// TwinCAT 3 PLC project PLC
// ProgramVersion: 3.1.4024.0
// libraries:
//   Tc2_EtherCAT, * (Beckhoff Automation GmbH)
//   Tc2_Standard, * (Beckhoff Automation GmbH)
//   Tc2_System, * (Beckhoff Automation GmbH)
//   Tc3_Module, * (Beckhoff Automation GmbH)
//   VisuDialogs, * (System)
// project tree:
//   DUTs/ ST_3D_Values.TcDUT
//   / GlobalTextList.TcGTLO, PlcTask.TcTTO, Visualisierungsmanager.TcVMO (not stored)
//   GVLs/ GVL_SensorFusion.TcGVL
//   POUs/Filter/ FB_ComplementaryFilter.TcPOU, FB_KalmanFilter.TcPOU, FB_MadgwickFilter.TcPOU, FB_MahonyFilter.TcPOU, FB_MovingAverageFilter.TcPOU (not stored), FB_MovingAverageFilter_3D.TcPOU
//   POUs/Filter/obsolete/ FBiFilter.TcPOU (not stored), FB_Complementary_Ex.TcPOU
//   POUs/Helping Functions/ ATAN2.TcPOU, ATAN2_deg.TcPOU
//   POUs/Helping Functions/obsolete/ iGetNextBufferPointer.TcPOU, iGetPriorBufferPointer.TcPOU
//   POUs/ MAIN.TcPOU
//   VISUs/ Visualization.TcVIS
// real-time tasks:
//   TASK PlcTask: cycle T#250us, priority 20, ADS port 350
// I/O:
//   DEVICE Device 3 (EtherCAT) (disabled), AmsNetId 172.17.129.121.4.1
//     Box 1 (EP3751-0260) [EP3751-0260 Acceleration Sensor and Gyroscope]
// variable links:
//   PLC/PLC Instance <-> Device 3 (EtherCAT)/Box 1 (EP3751-0260)
//     PlcTask Inputs/MAIN.stAccAxis/X <-> AI Acc X Samples 1 (Real32)/Samples[0]
//     PlcTask Inputs/MAIN.stAccAxis/Y <-> AI Acc Y Samples 1 (Real32)/Samples[0]
//     PlcTask Inputs/MAIN.stAccAxis/Z <-> AI Acc Z Samples 1 (Real32)/Samples[0]
//     PlcTask Inputs/MAIN.stGyroAxis/X <-> AI Gyro X Samples 1 (Real32)/Samples[0]
//     PlcTask Inputs/MAIN.stGyroAxis/Y <-> AI Gyro Y Samples 1 (Real32)/Samples[0]
//     PlcTask Inputs/MAIN.stGyroAxis/Z <-> AI Gyro Z Samples 1 (Real32)/Samples[0]

CONFIGURATION PLC
    RESOURCE PLC ON TwinCAT3
        TASK PlcTask(INTERVAL := T#250us, PRIORITY := 20);
        PROGRAM MAIN WITH PlcTask : MAIN;
    END_RESOURCE
END_CONFIGURATION

// ---- DUTs/ST_3D_Values.TcDUT
TYPE ST_3D_Values :
STRUCT
	X :REAL;
	Y :REAL;
	Z :REAL;
END_STRUCT
END_TYPE

// ---- GVLs/GVL_SensorFusion.TcGVL
{attribute 'qualified_only'}
VAR_GLOBAL CONSTANT
	buffersize_filter :UINT :=2000;
END_VAR

// ---- POUs/MAIN.TcPOU
PROGRAM MAIN
VAR
	stGyroAxis AT %I* : ST_3d_values;
	stcorrAxis : ST_3d_values;
	stOffset	:ST_3d_values;

	fbMovingAverage_3D: FB_MovingAverageFilter_3D;
	a_fBuffer : ARRAY[0..2] OF ARRAY[ 0..GVL_SensorFusion.buffersize_filter-1] OF REAL;
	
(* Accelerometer values *)
	stAccAxis AT %I* : ST_3d_values;
	normalizedAcceleration : ARRAY [0..2] OF LREAL;

(* Working variables *)
	fbStartOffsetCalibration : R_TRIG;
	bReset: BOOL;
	fbOffsetSet : R_TRIG;
	bResetAngles: BOOL;

	fCycleTime 				: LREAL; // PLC cycle time in s (has to match with ODR of sensor => for prototype this is static 4000Hz)
	nTaskIndex				: DINT;
	bReady					: BOOL;
	
(*Disclaimer: This is a sample still in prototype phase.
Please be aware that functionalities/ PDOs / CoEs can differ in series variant.
*)
	fbKalmanFilter:FB_KalmanFilter;
	fbMadgwickFilter:FB_MadgwickFilter;
	fbComplementaryFilter:FB_ComplementaryFilter;
	fbMahonyFilter:FB_MahonyFilter;
	stEulerAngle_Gyro:ST_3D_Values;
END_VAR

nTaskIndex:=GETCURTASKINDEXEX();
IF nTaskIndex>0 THEN
	fCycletime:=UDINT_TO_LREAL(_TaskInfo[GETCURTASKINDEXEX()].CycleTime) / 10_000_000;
END_IF

// get Sensoroffset
fbStartOffsetCalibration(clk:=bReset);

fbMovingAverage_3D( stSampleData:=stGyroAxis, bEnable:=NOT fbStartOffsetCalibration.Q, a_fSamples:=a_fBuffer);
fbOffsetSet(clk:=fbMovingAverage_3D.bBufferFilledX);
IF fbOffsetSet.Q THEN
	stOffset.x:=fbMovingAverage_3D.stAvgData.X;
	stOffset.y:=fbMovingAverage_3D.stAvgData.y;
	stOffset.z:=fbMovingAverage_3D.stAvgData.z;
	stEulerAngle_Gyro.x:=0;
	stEulerAngle_Gyro.y:=0;
	stEulerAngle_Gyro.z:=0;
ELSIF bResetAngles THEN
	stEulerAngle_Gyro.x:=0;
	stEulerAngle_Gyro.y:=0;
	stEulerAngle_Gyro.z:=0;
	bResetAngles:=FALSE;
END_IF

bReady:=fbMovingAverage_3D.bBufferFilledX;

//correct Gyro-Values with Offset
stcorrAxis.X:= stGyroAxis.X - stOffset.x;
stcorrAxis.Y:= stGyroAxis.Y - stOffset.y;
stcorrAxis.Z:= stGyroAxis.Z - stOffset.z;


	//Calculate Euler Angles by Sensorfusion
	fbKalmanFilter(
		stAccelData:= stAccAxis, 
		stGyroData:= stcorrAxis,  
		fCycleTime:= fCycletime,
		bSetReference:=fbMovingAverage_3D.bBufferFilledX );
		
	fbMadgwickFilter(
		stAccelData:= stAccAxis, 
		stGyroData:= stcorrAxis,  
		fcycletime:=fCycletime , 
		bSetReference:= fbMovingAverage_3D.bBufferFilledX );
		
	fbComplementaryFilter(
		stAccelData:= stAccAxis, 
		stGyroData:= stcorrAxis,  
		fcycletime:=fCycletime , 
		bSetReference:= fbMovingAverage_3D.bBufferFilledX );
		
	fbMahonyFilter(
		stAccelData:= stAccAxis, 
		stGyroData:= stcorrAxis,  
		fcycletime:=fCycletime , 
		bSetReference:= fbMovingAverage_3D.bBufferFilledX );
		
stEulerAngle_Gyro.x := stEulerAngle_Gyro.x + stcorrAxis.x * fCycleTime;
stEulerAngle_Gyro.y := stEulerAngle_Gyro.y + stcorrAxis.y * fCycleTime;
stEulerAngle_Gyro.z := stEulerAngle_Gyro.z + stcorrAxis.Z * fCycleTime;

END_PROGRAM

// ---- POUs/Filter/FB_MovingAverageFilter_3D.TcPOU
FUNCTION_BLOCK FB_MovingAverageFilter_3D
VAR_INPUT
    stSampleData : ST_3D_values; // New Data in 3 axes
    nNumSamples : UINT:= gvl_sensorFusion.buffersize_filter;              // Number of samples for the moving average
    bEnable 	: BOOL;                   // Execute flag
END_VAR

VAR_OUTPUT
    stAvgData : ST_3D_values; // New Data in 3 axes
    bBufferFilledX : BOOL;            // Flag indicating if the buffer for X axis is filled
    bBufferFilledY : BOOL;            // Flag indicating if the buffer for Y axis is filled
    bBufferFilledZ : BOOL;            // Flag indicating if the buffer for Z axis is filled
END_VAR

VAR_IN_OUT
    a_fSamples : ARRAY[0..2] OF ARRAY[ 0..GVL_SensorFusion.buffersize_filter-1] OF REAL; // Array of arrays to store samples for three axes
END_VAR

VAR
	fbExecuteTrigger:r_trig;
	bInit:BOOL;
    fbMovingAverageX : FB_MovingAverageFilter; // Instance for X axis
    fbMovingAverageY : FB_MovingAverageFilter; // Instance for Y axis
    fbMovingAverageZ : FB_MovingAverageFilter; // Instance for Z axis
END_VAR

IF NOT bEnable THEN
	bInit:=bInit;
END_IF

fbMovingAverageX(
    fInputValue := stSampleData.X,
    nNumSamples := nNumSamples,
    bEnable := bEnable,
    fAvgValue => stAvgData.x,
    bBufferFilled => bBufferFilledX,
    a_fSamples := a_fSamples[0]
);

fbMovingAverageY(
    fInputValue := stSampleData.y,
    nNumSamples := nNumSamples,
    bEnable := bEnable,
    fAvgValue => stAvgData.y,
    bBufferFilled => bBufferFilledY,
    a_fSamples := a_fSamples[1]
);

fbMovingAverageZ(
    fInputValue := stSampleData.z,
    nNumSamples := nNumSamples,
    bEnable := bEnable,
    fAvgValue => stAvgData.z,
    bBufferFilled => bBufferFilledZ,
    a_fSamples := a_fSamples[2]
);

END_FUNCTION_BLOCK

// ---- POUs/Filter/FB_KalmanFilter.TcPOU
FUNCTION_BLOCK FB_KalmanFilter
VAR_INPUT
    stAccelData : ST_3D_values; // Acceleration Data in (g)
    stGyroData : ST_3D_values; // Gyroscope Data in (°/s)
	fCycleTime: REAL; 			// CycleTime of sensor data in s
	fQ_angle : REAL := 0.001;     // Process noise variance for the angle
    fQ_bias : REAL := 0.003;      // Process noise variance for the bias
    fR_measure : REAL := 0.03;    // Measurement noise variance
    bSetReference : BOOL := FALSE; // Flag to set the current position as the reference position
END_VAR
VAR_OUTPUT
    stEulerAngle_deg : ST_3D_values; // Estimated Euler angle in degrees X= Pitch, Y=Roll, Z=Yaw
    stEulerAngle_rad : ST_3D_values; // Estimated Euler angle in rad X= Pitch, Y=Roll, Z=Yaw
END_VAR
VAR
	// Reference angles
	stRef_Angles_deg :ST_3d_values; // Reference orientation (bSetReference; angles in degrees)
	
    // Variables for X-axis
    fAngle_prevX_rad : LREAL := 0.0;   // Previous angle for X-axis in radians
    fBiasX : LREAL := 0.0;             // Gyroscope bias for X-axis
    fRateX : LREAL := 0.0;             // Rate of change of the angle for X-axis

    fP_00X : LREAL := 1.0;             // Covariance matrix for X-axis
    fP_01X : LREAL := 0.0;
    fP_10X : LREAL := 0.0;
    fP_11X : LREAL := 1.0;

    fY_X : LREAL;                      // Angle difference for X-axis
    fS_X : LREAL;                      // Estimate error for X-axis
    fK_0X : LREAL;                     // Kalman gain for X-axis
    fK_1X : LREAL;                     // Kalman gain for X-axis

    // Variables for Y-axis
    fAngle_prevY_rad : LREAL := 0.0;   // Previous angle for Y-axis in radians
    fBiasY : LREAL := 0.0;             // Gyroscope bias for Y-axis
    fRateY : LREAL := 0.0;             // Rate of change of the angle for Y-axis

    fP_00Y : LREAL := 1.0;             // Covariance matrix for Y-axis
    fP_01Y : LREAL := 0.0;
    fP_10Y : LREAL := 0.0;
    fP_11Y : LREAL := 1.0;

    fY_Y : LREAL;                      // Angle difference for Y-axis
    fS_Y : LREAL;                      // Estimate error for Y-axis
    fK_0Y : LREAL;                     // Kalman gain for Y-axis
    fK_1Y : LREAL;                     // Kalman gain for Y-axis

    // Variables for Z-axis
    fAngle_prevZ_rad : LREAL := 0.0;   // Previous angle for Z-axis in radians
    fBiasZ : LREAL := 0.0;             // Gyroscope bias for Z-axis
    fRateZ : LREAL := 0.0;             // Rate of change of the angle for Z-axis

    fP_00Z : LREAL := 1.0;             // Covariance matrix for Z-axis
    fP_01Z : LREAL := 0.0;
    fP_10Z : LREAL := 0.0;
    fP_11Z : LREAL := 1.0;

    fY_Z : LREAL;                      // Angle difference for Z-axis
    fS_Z : LREAL;                      // Estimate error for Z-axis
    fK_0Z : LREAL;                     // Kalman gain for Z-axis
    fK_1Z : LREAL;                     // Kalman gain for Z-axis
	
	// Convert accelerometer data to angles (pitch, roll) in radians
    fPitchAccel_rad : LREAL;
    fRollAccel_rad : LREAL;
	
	fbSetReference: r_trig;
END_VAR

// Calculate accelerometer angles using ATAN2, which returns radians
IF (stAccelData.X * stAccelData.X + stAccelData.Z * stAccelData.Z > 0.0) THEN 
    fPitchAccel_rad := ATAN(stAccelData.Y / SQRT(stAccelData.X * stAccelData.X + stAccelData.Z * stAccelData.Z));
END_IF
IF (stAccelData.Y * stAccelData.Y + stAccelData.Z * stAccelData.Z > 0.0) THEN 
    fRollAccel_rad := ATAN(stAccelData.X / SQRT(stAccelData.Y * stAccelData.Y + stAccelData.Z * stAccelData.Z));
END_IF

// Prediction step for X-axis (Pitch)
fRateX := stGyroData.X - fBiasX;
fAngle_prevX_rad := fAngle_prevX_rad + fCycleTime * fRateX * PI / 180.0; // Conversion of rate from degrees/second to radians/second

fP_00X := fP_00X + fCycleTime * (fCycleTime * fP_11X - fP_01X - fP_10X + fQ_angle);
fP_01X := fP_01X - fCycleTime * fP_11X;
fP_10X := fP_10X - fCycleTime * fP_11X;
fP_11X := fP_11X + fQ_bias * fCycleTime;

// Measurement update for X-axis (Pitch)
fY_X := fPitchAccel_rad - fAngle_prevX_rad; // Using the pitch angle in radians
fS_X := fP_00X + fR_measure;
fK_0X := fP_00X / fS_X;
fK_1X := fP_10X / fS_X;

fAngle_prevX_rad := fAngle_prevX_rad + fK_0X * fY_X;
fBiasX := fBiasX + fK_1X * fY_X;

fP_00X := fP_00X - fK_0X * fP_00X;
fP_01X := fP_01X - fK_0X * fP_01X;
fP_10X := fP_10X - fK_1X * fP_00X;
fP_11X := fP_11X - fK_1X * fP_01X;

// Prediction step for Y-axis (Roll)
fRateY := stGyroData.Y - fBiasY;
fAngle_prevY_rad := fAngle_prevY_rad + fCycleTime * fRateY * PI / 180.0; // Conversion of rate from degrees/second to radians/second

fP_00Y := fP_00Y + fCycleTime * (fCycleTime * fP_11Y - fP_01Y - fP_10Y + fQ_angle);
fP_01Y := fP_01Y - fCycleTime * fP_11Y;
fP_10Y := fP_10Y - fCycleTime * fP_11Y;
fP_11Y := fP_11Y + fQ_bias * fCycleTime;

// Measurement update for Y-axis (Roll)
fY_Y := fRollAccel_rad - fAngle_prevY_rad; // Using the roll angle in radians
fS_Y := fP_00Y + fR_measure;
fK_0Y := fP_00Y / fS_Y;
fK_1Y := fP_10Y / fS_Y;

fAngle_prevY_rad := fAngle_prevY_rad + fK_0Y * fY_Y;
fBiasY := fBiasY + fK_1Y * fY_Y;

fP_00Y := fP_00Y - fK_0Y * fP_00Y;
fP_01Y := fP_01Y - fK_0Y * fP_01Y;
fP_10Y := fP_10Y - fK_1Y * fP_00Y;
fP_11Y := fP_11Y - fK_1Y * fP_01Y;

// Prediction step for Z-axis (Yaw)
fRateZ := stGyroData.Z - fBiasZ;
fAngle_prevZ_rad := fAngle_prevZ_rad + fCycleTime * fRateZ * PI / 180.0; // Conversion of rate from degrees/second to radians/second

fP_00Z := fP_00Z + fCycleTime * (fCycleTime * fP_11Z - fP_01Z - fP_10Z + fQ_angle);
fP_01Z := fP_01Z - fCycleTime * fP_11Z;
fP_10Z := fP_10Z - fCycleTime * fP_11Z;
fP_11Z := fP_11Z + fQ_bias * fCycleTime;

// Measurement update for Z-axis (Yaw)
// Since the accelerometer does not provide a direct yaw measurement, we use gyroscope data for the yaw update.
fY_Z := fRateZ; // Gyroscope rate in degrees/second
fS_Z := fP_00Z + fR_measure;
fK_0Z := fP_00Z / fS_Z;
fK_1Z := fP_10Z / fS_Z;

fAngle_prevZ_rad := fAngle_prevZ_rad + fK_0Z * fY_Z * fCycleTime * PI / 180.0; // Updating the yaw angle with gyroscope data and conversion to radians
fBiasZ := fBiasZ + fK_1Z * fY_Z * fCycleTime * PI / 180.0;

fP_00Z := fP_00Z - fK_0Z * fP_00Z;
fP_01Z := fP_01Z - fK_0Z * fP_01Z;
fP_10Z := fP_10Z - fK_1Z * fP_00Z;
fP_11Z := fP_11Z - fK_1Z * fP_01Z;

// Convert radians to degrees for output
stEulerAngle_deg.X := fAngle_prevX_rad * 180.0 / PI;
stEulerAngle_deg.Y := fAngle_prevY_rad * 180.0 / PI;
stEulerAngle_deg.Z := fAngle_prevZ_rad * 180.0 / PI;

fbSetReference(clk:=bSetReference);
// Set reference position if flag is active
IF fbSetReference.q THEN
    stRef_Angles_deg.X := stEulerAngle_deg.X;
    stRef_Angles_deg.Y := stEulerAngle_deg.Y;
    stRef_Angles_deg.Z := stEulerAngle_deg.Z;
END_IF

// Apply reference position
stEulerAngle_deg.X := stEulerAngle_deg.X - (stRef_Angles_deg.X);
stEulerAngle_deg.Y := stEulerAngle_deg.Y - (stRef_Angles_deg.Y);
stEulerAngle_deg.Z := stEulerAngle_deg.Z - (stRef_Angles_deg.Z);

stEulerAngle_rad.X := fAngle_prevX_rad - (stRef_Angles_deg.X) * PI / 180.0;
stEulerAngle_rad.Y := fAngle_prevY_rad - (stRef_Angles_deg.Y) * PI / 180.0;
stEulerAngle_rad.Z := fAngle_prevZ_rad - (stRef_Angles_deg.Z) * PI / 180.0;

END_FUNCTION_BLOCK

// ---- POUs/Filter/FB_MadgwickFilter.TcPOU
FUNCTION_BLOCK FB_MadgwickFilter
VAR_INPUT
    stAccelData : ST_3D_values; // Acceleration Data in (g)
    stGyroData : ST_3D_values; // Gyroscope Data in (°/s)
    fBeta: REAL := 0.05; // Algorithm gain
    fCycletime: REAL; // Time step (s)
    bSetReference: BOOL; // Flag to set reference position
END_VAR

VAR_OUTPUT
	fQ0 : LREAL := 1.0; // Quaternion component
    fQ1 : LREAL := 0.0; // Quaternion component
    fQ2 : LREAL := 0.0; // Quaternion component
    fQ3 : LREAL := 0.0; // Quaternion component
    stEulerAngle_deg : ST_3D_values; // Estimated Euler angle in degrees X= Pitch, Y=Roll, Z=Yaw
    stEulerAngle_rad : ST_3D_values; // Estimated Euler angle in rad X= Pitch, Y=Roll, Z=Yaw
END_VAR

VAR

	// Reference angles
	stRef_Angles_deg :ST_3d_values; // Reference orientation (bSetReference; angles in degrees)
    fNorm : LREAL;
    _2fQ0, _2fQ1, _2fQ2, _2fQ3 : LREAL;
    _4fQ0, _4fQ1, _4fQ2, _4fQ3 : LREAL;
    _8fQ1, _8fQ2 : LREAL;
    fQ0fQ0, fQ1fQ1, fQ2fQ2, fQ3fQ3 : LREAL;
    fAx, fAy, fAz : LREAL;
    fS1, fS2, fS3, fS4 : LREAL;
    fSinRoll, fCosRoll : LREAL;
    fSinPitch, fCosPitch : LREAL;
    fSinYaw, fCosYaw : LREAL;
	fGyroRateX_rad,fGyroRateY_rad, fGyroRateZ_rad:LREAL;
	fbSetReference: r_trig;
END_VAR

// Normalize accelerometer measurements
fAx := REAL_TO_LREAL(stAccelData.x);
fAy := REAL_TO_LREAL(stAccelData.y);
fAz := REAL_TO_LREAL(stAccelData.z);
fNorm := fAx * fAx + fAy * fAy + fAz * fAz;
IF fNorm > 1E-6 THEN
    fNorm := SQRT(fNorm);
    fAx := fAx / fNorm;
    fAy := fAy / fNorm;
    fAz := fAz / fNorm;
END_IF

// Estimated direction of gravity and magnetic field
_2fQ0 := 2.0 * fQ0;
_2fQ1 := 2.0 * fQ1;
_2fQ2 := 2.0 * fQ2;
_2fQ3 := 2.0 * fQ3;
_4fQ0 := 4.0 * fQ0;
_4fQ1 := 4.0 * fQ1;
_4fQ2 := 4.0 * fQ2;
_4fQ3 := 4.0 * fQ3;
_8fQ1 := 8.0 * fQ1;
_8fQ2 := 8.0 * fQ2;
fQ0fQ0 := fQ0 * fQ0;
fQ1fQ1 := fQ1 * fQ1;
fQ2fQ2 := fQ2 * fQ2;
fQ3fQ3 := fQ3 * fQ3;

// Gradient descent algorithm corrective step
fS1 := _4fQ0 * fQ2fQ2 + _2fQ2 * fAx + _4fQ0 * fQ1fQ1 - _2fQ1 * fAy;
fS2 := _4fQ1 * fQ3fQ3 - _2fQ3 * fAx + 4.0 * fQ0fQ0 * fQ1 - _2fQ0 * fAy - _4fQ1 + _8fQ1 * fQ1fQ1 + _8fQ1 * fQ2fQ2 + _4fQ1 * fAz;
fS3 := 4.0 * fQ0fQ0 * fQ2 + _2fQ0 * fAx + _4fQ2 * fQ3fQ3 - _2fQ3 * fAy - _4fQ2 + _8fQ2 * fQ1fQ1 + _8fQ2 * fQ2fQ2 + _4fQ2 * fAz;
fS4 := 4.0 * fQ1fQ1 * fQ3 - _2fQ1 * fAx + 4.0 * fQ2fQ2 * fQ3 - _2fQ2 * fAy;

// Normalize step magnitude
fNorm := fS1 * fS1 + fS2 * fS2 + fS3 * fS3 + fS4 * fS4;
IF fNorm > 1E-6 THEN
    fNorm := SQRT(fNorm);
    fS1 := fS1 / fNorm;
    fS2 := fS2 / fNorm;
    fS3 := fS3 / fNorm;
    fS4 := fS4 / fNorm;
END_IF

// Apply gradient descent corrective step
fQ0 := fQ0 - REAL_TO_LREAL(fBeta) * fS1 * REAL_TO_LREAL(fCycleTime);
fQ1 := fQ1 - REAL_TO_LREAL(fBeta) * fS2 * REAL_TO_LREAL(fCycleTime);
fQ2 := fQ2 - REAL_TO_LREAL(fBeta) * fS3 * REAL_TO_LREAL(fCycleTime);
fQ3 := fQ3 - REAL_TO_LREAL(fBeta) * fS4 * REAL_TO_LREAL(fCycleTime);

// Convert gyroscope rates from °/s to rad/s
fGyroRateX_rad := stGyroData.x * pi / 180.0;
fGyroRateY_rad := stGyroData.y * pi / 180.0;
fGyroRateZ_rad := stGyroData.z * pi / 180.0;

// Integrate rate of change of quaternion
fQ0 := fQ0 + 0.5 * (-fQ1 * REAL_TO_LREAL(fGyroRateX_rad) - fQ2 * REAL_TO_LREAL(fGyroRateY_rad) - fQ3 * REAL_TO_LREAL(fGyroRateZ_rad)) * REAL_TO_LREAL(fCycleTime);
fQ1 := fQ1 + 0.5 * (fQ0 * REAL_TO_LREAL(fGyroRateX_rad) + fQ2 * REAL_TO_LREAL(fGyroRateZ_rad) - fQ3 * REAL_TO_LREAL(fGyroRateY_rad)) * REAL_TO_LREAL(fCycleTime);
fQ2 := fQ2 + 0.5 * (fQ0 * REAL_TO_LREAL(fGyroRateY_rad) - fQ1 * REAL_TO_LREAL(fGyroRateZ_rad) + fQ3 * REAL_TO_LREAL(fGyroRateX_rad)) * REAL_TO_LREAL(fCycleTime);
fQ3 := fQ3 + 0.5 * (fQ0 * REAL_TO_LREAL(fGyroRateZ_rad) + fQ1 * REAL_TO_LREAL(fGyroRateY_rad) - fQ2 * REAL_TO_LREAL(fGyroRateX_rad)) * REAL_TO_LREAL(fCycleTime);

// Normalize quaternion
fNorm := fQ0 * fQ0 + fQ1 * fQ1 + fQ2 * fQ2 + fQ3 * fQ3;
IF fNorm > 1E-6 THEN
    fNorm := SQRT(fNorm);
    fQ0 := fQ0 / fNorm;
    fQ1 := fQ1 / fNorm;
    fQ2 := fQ2 / fNorm;
    fQ3 := fQ3 / fNorm;
END_IF

// Calculate trigonometric values directly from quaternion components
fSinRoll := 2.0 * (fQ0 * fQ1 + fQ2 * fQ3);
fCosRoll := 1.0 - 2.0 * (fQ1 * fQ1 + fQ2 * fQ2);
fSinPitch := 2.0 * (fQ0 * fQ2 - fQ3 * fQ1);
fCosPitch := 1.0 - 2.0 * (fQ2 * fQ2 + fQ3 * fQ3);
fSinYaw := 2.0 * (fQ0 * fQ3 + fQ1 * fQ2);
fCosYaw := 1.0 - 2.0 * (fQ3 * fQ3 + fQ2 * fQ2);

// Convert trigonometric values to Euler angles using ATAN2 and ASIN in radians
stEulerAngle_rad.x := LREAL_TO_REAL(ATAN2(fSinRoll, fCosRoll));
stEulerAngle_rad.y := LREAL_TO_REAL(ASIN(fSinPitch));
stEulerAngle_rad.Z := LREAL_TO_REAL(ATAN2(fSinYaw, fCosYaw));

// Convert radians to degrees
stEulerAngle_deg.x := stEulerAngle_rad.x * 180.0 / pi;
stEulerAngle_deg.y := stEulerAngle_rad.y * 180.0 / pi;
stEulerAngle_deg.z := stEulerAngle_rad.z * 180.0 / pi;

fbSetReference(clk:=bSetReference);
// Set reference position if flag is active
IF fbSetReference.q THEN
    stRef_Angles_deg.X := stEulerAngle_deg.X;
    stRef_Angles_deg.Y := stEulerAngle_deg.Y;
    stRef_Angles_deg.Z := stEulerAngle_deg.Z;
END_IF

// Apply reference position
stEulerAngle_deg.X := stEulerAngle_deg.X - (stRef_Angles_deg.X);
stEulerAngle_deg.Y := stEulerAngle_deg.Y - (stRef_Angles_deg.Y);
stEulerAngle_deg.Z := stEulerAngle_deg.Z - (stRef_Angles_deg.Z);

stEulerAngle_rad.X := stEulerAngle_rad.X - (stRef_Angles_deg.X) * PI / 180.0;
stEulerAngle_rad.Y := stEulerAngle_rad.Y - (stRef_Angles_deg.Y) * PI / 180.0;
stEulerAngle_rad.Z := stEulerAngle_rad.Z - (stRef_Angles_deg.Z) * PI / 180.0;

END_FUNCTION_BLOCK

// ---- POUs/Helping Functions/ATAN2.TcPOU
FUNCTION ATAN2 : LREAL //in rad
VAR_INPUT	
    y : REAL; // y-coordinate
    x : REAL; // x-coordinate
END_VAR
VAR_OUTPUT
   
END_VAR

IF x > 0 THEN
    ATAN2 := ATAN(y / x);
ELSIF x < 0 AND y >= 0 THEN
    ATAN2 := ATAN(y / x) + pi;
ELSIF x < 0 AND y < 0 THEN
    ATAN2 := ATAN(y / x) - pi;
ELSIF x = 0 AND y > 0 THEN
    ATAN2 := pi / 2;
ELSIF x = 0 AND y < 0 THEN
    ATAN2 := -pi / 2;
ELSIF x = 0 AND y = 0 THEN
    ATAN2 := 0.0; // Undefined, but conventionally set to 0
END_IF

END_FUNCTION

// ---- POUs/Filter/FB_ComplementaryFilter.TcPOU
FUNCTION_BLOCK FB_ComplementaryFilter
VAR_INPUT
    stAccelData : ST_3D_values; // Acceleration Data in (g)
    stGyroData : ST_3D_values; // Gyroscope Data in (°/s)
    fCycleTime : REAL; // Cycle Time (s)
    fAlpha : REAL := 0.98; // Filter coefficient
    bSetReference : BOOL; // Flag to set reference position
END_VAR

VAR_OUTPUT
    stEulerAngle_deg : ST_3D_values; // Euler angle in degrees X= Pitch, Y=Roll, Z=Yaw
    stEulerAngle_rad : ST_3D_values; // Euler angle in rad X= Pitch, Y=Roll, Z=Yaw
END_VAR

VAR
	stRef_Angles_deg :ST_3d_values; // Reference orientation (bSetReference; angles in degrees)
	
    fAccAngleRoll : REAL;
    fAccAnglePitch : REAL;
	
    fGyroAngleRoll : REAL;
    fGyroAnglePitch : REAL;
    fGyroAngleYaw : REAL;
	
	fbSetReference: r_trig;
END_VAR

// Calculate accelerometer angles using ATAN2, which returns radians
IF ((stAccelData.X * stAccelData.X + stAccelData.Z * stAccelData.Z)> 0.0) THEN 	
	fAccAngleRoll := ATAN2(stAccelData.Y, SQRT(stAccelData.X * stAccelData.X + stAccelData.Z * stAccelData.Z));
END_IF
IF ((stAccelData.Y * stAccelData.Y + stAccelData.Z * stAccelData.Z)> 0.0) THEN
	fAccAnglePitch := ATAN2(-stAccelData.X, SQRT(stAccelData.Y * stAccelData.Y + stAccelData.Z * stAccelData.Z));
END_IF

// Convert gyroscope rates from °/s to rad/s before integration
stGyroData.X := stGyroData.X * pi / 180.0;
stGyroData.Y := stGyroData.Y * pi / 180.0;
stGyroData.Z := stGyroData.Z * pi / 180.0;

// Integrate gyroscope rates to get angles in radians
fGyroAnglePitch := fGyroAnglePitch + stGyroData.X * fCycleTime;
fGyroAngleRoll := fGyroAngleRoll + stGyroData.Y * fCycleTime;
fGyroAngleYaw := fGyroAngleYaw + stGyroData.Z * fCycleTime;

// Apply complementary filter
stEulerAngle_rad.X := fAlpha * (fGyroAnglePitch) + (1.0 - fAlpha) * fAccAnglePitch;
stEulerAngle_rad.Y := fAlpha * (fGyroAngleRoll) + (1.0 - fAlpha) * fAccAngleRoll;
stEulerAngle_rad.Z := fGyroAngleYaw; // Yaw is integrated directly from gyroscope

// Convert radians to degrees for output
stEulerAngle_deg.X := stEulerAngle_rad.X * 180.0 / pi;
stEulerAngle_deg.Y := stEulerAngle_rad.Y * 180.0 / pi;
stEulerAngle_deg.Z := stEulerAngle_rad.Z * 180.0 / pi;

fbSetReference(clk:=bSetReference);
// Set reference position if flag is active
IF fbSetReference.q THEN
    stRef_Angles_deg.X := stEulerAngle_deg.X;
    stRef_Angles_deg.Y := stEulerAngle_deg.Y;
    stRef_Angles_deg.Z := stEulerAngle_deg.Z;
END_IF

// Apply reference position
stEulerAngle_deg.X := stEulerAngle_deg.X - (stRef_Angles_deg.X);
stEulerAngle_deg.Y := stEulerAngle_deg.Y - (stRef_Angles_deg.Y);
stEulerAngle_deg.Z := stEulerAngle_deg.Z- (stRef_Angles_deg.Z);

stEulerAngle_rad.X := stEulerAngle_rad.X - (stRef_Angles_deg.X) * pi / 180.0;
stEulerAngle_rad.Y := stEulerAngle_rad.Y - (stRef_Angles_deg.Y) * pi / 180.0;
stEulerAngle_rad.Z := stEulerAngle_rad.Z - (stRef_Angles_deg.Z) * pi / 180.0;

END_FUNCTION_BLOCK

// ---- POUs/Filter/FB_MahonyFilter.TcPOU
FUNCTION_BLOCK FB_MahonyFilter
VAR_INPUT
    stAccelData : ST_3D_values; // Acceleration Data in (g)
    stGyroData : ST_3D_values; // Gyroscope Data in (°/s)
    fCycleTime : REAL; // Cycle Time (s)
    fKp : REAL := 1.0; // Proportional gain
    fKi : REAL := 0.01; // Integral gain
    bSetReference : BOOL; // Flag to set reference position
END_VAR

VAR_OUTPUT
	fQ0 : LREAL := 1.0; // Quaternion component
    fQ1 : LREAL := 0.0; // Quaternion component
    fQ2 : LREAL := 0.0; // Quaternion component
    fQ3 : LREAL := 0.0; // Quaternion component
    stEulerAngle_deg : ST_3D_values; // Estimated Euler angle in degrees X= Pitch, Y=Roll, Z=Yaw
    stEulerAngle_rad : ST_3D_values; // Estimated Euler angle in rad X= Pitch, Y=Roll, Z=Yaw
END_VAR

VAR
	// Reference angles
	stRef_Angles_deg :ST_3d_values; // Reference orientation (bSetReference; angles in degrees)
    fIntegralFBx : LREAL := 0.0; // Integral feedback x
    fIntegralFBy : LREAL := 0.0; // Integral feedback y
    fIntegralFBz : LREAL := 0.0; // Integral feedback z
    fNorm : LREAL;
    _2fQ0, _2fQ1, _2fQ2, _2fQ3 : LREAL;
    _4fQ0, _4fQ1, _4fQ2, _4fQ3 : LREAL;
    _8fQ1, _8fQ2 : LREAL;
    fQ0fQ0, fQ1fQ1, fQ2fQ2, fQ3fQ3 : LREAL;
    fAx, fAy, fAz : LREAL;
    fEx, fEy, fEz : LREAL;
	fSinRoll, fCosRoll : LREAL;
    fSinPitch, fCosPitch : LREAL;
    fSinYaw, fCosYaw : LREAL;
	fGyroRateX_rad,fGyroRateY_rad, fGyroRateZ_rad:LREAL;
	
	q0, q1, q2, q3 :LREAL;
	q0n, q1n, q2n, q3n :LREAL;
	fbSetReference: r_trig;
END_VAR

// Normalize accelerometer measurements
fAx := REAL_TO_LREAL(stAccelData.x);
fAy := REAL_TO_LREAL(stAccelData.Y);
fAz := REAL_TO_LREAL(stAccelData.z);
fNorm := (fAx * fAx + fAy * fAy + fAz * fAz);
IF fNorm > 1E-6 THEN
    fNorm := SQRT(fNorm);
    fAx := fAx / fNorm;
    fAy := fAy / fNorm;
    fAz := fAz / fNorm;
END_IF

// Estimated direction of gravity and magnetic field
_2fQ0 := 2.0 * fQ0;
_2fQ1 := 2.0 * fQ1;
_2fQ2 := 2.0 * fQ2;
_2fQ3 := 2.0 * fQ3;
_4fQ0 := 4.0 * fQ0;
_4fQ1 := 4.0 * fQ1;
_4fQ2 := 4.0 * fQ2;
_4fQ3 := 4.0 * fQ3;
_8fQ1 := 8.0 * fQ1;
_8fQ2 := 8.0 * fQ2;
fQ0fQ0 := fQ0 * fQ0;
fQ1fQ1 := fQ1 * fQ1;
fQ2fQ2 := fQ2 * fQ2;
fQ3fQ3 := fQ3 * fQ3;

// Error is sum of cross product between estimated direction and measured direction of gravity
fEx := (_2fQ1 * fQ3 - _2fQ0 * fQ2) - fAx;
fEy := (_2fQ0 * fQ1 + _2fQ2 * fQ3) - fAy;
fEz := (_2fQ0 * fQ3 - _4fQ1 * fQ1 - _4fQ2 * fQ2) - fAz;

// Apply proportional feedback
stGyroData.x := stGyroData.x + REAL_TO_LREAL(fKp) * LREAL_TO_REAL(fEx);
stGyroData.y := stGyroData.y + REAL_TO_LREAL(fKp) * LREAL_TO_REAL(fEy);
stGyroData.z := stGyroData.z + REAL_TO_LREAL(fKp) * LREAL_TO_REAL(fEz);

// Convert gyroscope rates from °/s to rad/s
fGyroRateX_rad := stGyroData.x * pi / 180.0;
fGyroRateY_rad := stGyroData.y * pi / 180.0;
fGyroRateZ_rad := stGyroData.z * pi / 180.0;

// Integrate rate of change of quaternion
fQ0 := fQ0 + 0.5 * (-fQ1 * REAL_TO_LREAL(fGyroRateX_rad) - fQ2 * REAL_TO_LREAL(fGyroRateY_rad) - fQ3 * REAL_TO_LREAL(fGyroRateZ_rad)) * REAL_TO_LREAL(fCycleTime);
fQ1 := fQ1 + 0.5 * (fQ0 * REAL_TO_LREAL(fGyroRateX_rad) + fQ2 * REAL_TO_LREAL(fGyroRateZ_rad) - fQ3 * REAL_TO_LREAL(fGyroRateY_rad)) * REAL_TO_LREAL(fCycleTime);
fQ2 := fQ2 + 0.5 * (fQ0 * REAL_TO_LREAL(fGyroRateY_rad) - fQ1 * REAL_TO_LREAL(fGyroRateZ_rad) + fQ3 * REAL_TO_LREAL(fGyroRateX_rad)) * REAL_TO_LREAL(fCycleTime);
fQ3 := fQ3 + 0.5 * (fQ0 * REAL_TO_LREAL(fGyroRateZ_rad) + fQ1 * REAL_TO_LREAL(fGyroRateY_rad) - fQ2 * REAL_TO_LREAL(fGyroRateX_rad)) * REAL_TO_LREAL(fCycleTime);

// Normalize quaternion
fNorm := (fQ0 * fQ0 + fQ1 * fQ1 + fQ2 * fQ2 + fQ3 * fQ3);
IF fNorm > 1E-6 THEN
    fNorm := SQRT(fNorm);
    fQ0 := fQ0 / fNorm;
    fQ1 := fQ1 / fNorm;
    fQ2 := fQ2 / fNorm;
    fQ3 := fQ3 / fNorm;
END_IF

// Calculate trigonometric values directly from quaternion components
fSinRoll := 2.0 * (fQ0 * fQ1 + fQ2 * fQ3);
fCosRoll := 1.0 - 2.0 * (fQ1 * fQ1 + fQ2 * fQ2);
fSinPitch := 2.0 * (fQ0 * fQ2 - fQ3 * fQ1);
fCosPitch := 1.0 - 2.0 * (fQ2 * fQ2 + fQ3 * fQ3);
fSinYaw := 2.0 * (fQ0 * fQ3 + fQ1 * fQ2);
fCosYaw := 1.0 - 2.0 * (fQ3 * fQ3 + fQ2 * fQ2);

// Convert trigonometric values to Euler angles using ATAN2 and ASIN in radians
stEulerAngle_rad.x := LREAL_TO_REAL(ATAN2(fSinRoll, fCosRoll));
stEulerAngle_rad.y := LREAL_TO_REAL(ASIN(fSinPitch));
stEulerAngle_rad.Z := LREAL_TO_REAL(ATAN2(fSinYaw, fCosYaw));

// Convert radians to degrees
stEulerAngle_deg.x := stEulerAngle_rad.x * 180.0 / pi;
stEulerAngle_deg.y := stEulerAngle_rad.y * 180.0 / pi;
stEulerAngle_deg.z := stEulerAngle_rad.z * 180.0 / pi;

fbSetReference(clk:=bSetReference);
// Set reference position if flag is active
IF fbSetReference.q THEN
    stRef_Angles_deg.X := stEulerAngle_deg.X;
    stRef_Angles_deg.Y := stEulerAngle_deg.Y;
    stRef_Angles_deg.Z := stEulerAngle_deg.Z;
END_IF

// Apply reference position
stEulerAngle_deg.X := stEulerAngle_deg.X - (stRef_Angles_deg.X);
stEulerAngle_deg.Y := stEulerAngle_deg.Y - (stRef_Angles_deg.Y);
stEulerAngle_deg.Z := stEulerAngle_deg.Z - (stRef_Angles_deg.Z);

stEulerAngle_rad.X := stEulerAngle_rad.X - (stRef_Angles_deg.X) * PI / 180.0;
stEulerAngle_rad.Y := stEulerAngle_rad.Y - (stRef_Angles_deg.Y) * PI / 180.0;
stEulerAngle_rad.Z := stEulerAngle_rad.Z - (stRef_Angles_deg.Z) * PI / 180.0;

END_FUNCTION_BLOCK

// ---- POUs/Filter/obsolete/FB_Complementary_Ex.TcPOU
FUNCTION FB_Complementary_Ex : real
VAR_INPUT
    stAccelData : ST_3D_values; // Acceleration Data in (g)
    stGyroData : ST_3D_values; // Gyroscope Data in (°/s)
    fCycleTime : REAL; // Cycle Time (s)
    fAlpha : REAL := 0.98; // Filter coefficient
    bSetReference : BOOL; // Flag to set reference position
END_VAR
VAR
	   
	    fAccAngleRoll 	: REAL;
        fAccAnglePitch 	: REAL;
   
		fGyroAngleRoll : REAL;
    	fGyroAnglePitch : REAL;
    	fGyroAngleYaw : REAL;

		fIntegrator_Pitch 	: REAL;
	    fIntegrator_Roll : REAL;
        fIntegrator_Yaw 	: REAL;
		
		droll	: LREAL;
		dpitch	: LREAL;
		dyaw	: LREAL;
END_VAR


//	Deg[z] := fIntegrator_Pitch * 360.0;
fIntegrator_Pitch	:= fIntegrator_Pitch + (stAccelData.X * fCycleTime /360.0);
fIntegrator_Roll 	:= fIntegrator_Roll + (stAccelData.Y* fCycleTime /360.0);
fIntegrator_Yaw 	:= fIntegrator_Yaw + (stAccelData.Z* fCycleTime /360.0);



(* calculate the delta movements *)
droll := actualRoll;
dpitch := actualPitch;
dyaw := actualYaw;

actualRoll := fIntegrator_Pitch * 2 * PI;
actualPitch := fIntegrator_Roll * 2 * PI;
actualYaw := fIntegrator_Yaw * 2 * PI;

droll := actualRoll - droll;
dpitch := actualPitch - dpitch;
dyaw := actualYaw - dyaw;

(* Axis correction *)
dyaw := dyaw;
temp := dpitch;
dpitch := -droll;
droll := temp;

(* Calculate the euler speeds *)
fphi := droll + SIN(actualPhi)*TAN(actualTheta)*dpitch + COS(actualPhi)*TAN(actualTheta)*dyaw;
ftheta := COS(actualPhi)*dpitch-SIN(actualPhi)*dyaw;
fPsi := (SIN(actualPhi)/COS(actualTheta)) * dpitch + (COS(actualPhi)/COS(actualTheta))*dyaw;


(* Calculate new euler angles *)
actualPhi := actualPhi + fphi;
actualTheta := actualTheta + ftheta;
actualPsi := actualPsi + fPsi;

(* Collapse if passing thresholds of pi *)
IF actualPhi < 0 THEN actualPhi := actualPhi + 2*PI; END_IF
IF actualPhi >= 2*PI THEN actualPhi := actualPhi - 2*PI; END_IF
IF actualTheta < 0 THEN	actualTheta := actualTheta + 2*PI; END_IF
IF actualTheta >= 2*PI THEN	actualTheta := actualTheta - 2*PI; END_IF
IF actualPsi < 0 THEN	actualPsi := actualPsi + 2*PI;END_IF
IF actualPsi >= 2*PI THEN	actualPsi := actualPsi - 2*PI;END_IF

(* Determine length of acceleration vector *)
sumAcc := a_fAccAxis[0] * a_fAccAxis[0] + a_fAccAxis[1] * a_fAccAxis[1] + a_fAccAxis[2] * a_fAccAxis[2];
sumAcc := SQRT(sumAcc);

(* Normalize acceleration vector *)
IF sumAcc <> 0 THEN
	FOR z := 0 TO 2 DO
		normalizedAcceleration[z] := a_fAccAxis[z] / sumAcc;
	END_FOR
END_IF

(* Due to normalized values, we do no need to cut off higher values than 1 *)
IF normalizedAcceleration[2] = 0 THEN
	normalizedAcceleration[2] := 0.000001;
END_IF
AccPhi := -ATAN(normalizedAcceleration[0] / normalizedAcceleration[2]) + PI;
IF (a_fAccAxis[2]) <=0 THEN
	AccPhi := AccPhi + PI;
END_IF
IF AccPhi > 2*PI THEN AccPhi := AccPhi - 2*PI; END_IF;
IF AccPhi < 0 THEN AccPhi := AccPhi + 2*PI; END_IF;
AccTheta := ASIN(normalizedAcceleration[1]) + PI;
(* Simple sensor fusion if we are not accelerated *)
IF sumAcc >= (1.0 - fusionWindow) AND sumAcc <= (1.0 + fusionWindow)AND bUseSensorFusion THEN
	(* The AccPhi calculation is good, as long as Axis[2] ist not close to 0 *)
	IF normalizedAcceleration[2] < -fusionHorizontThreshold OR normalizedAcceleration[2] > fusionHorizontThreshold THEN
		IF (actualPhi - AccPhi) > PI OR (actualPhi - AccPhi) < -PI THEN
			IF AccPhi > actualPhi THEN
				AccPhi := AccPhi - 2 * PI;
			ELSE
				AccPhi := AccPhi + 2 * PI;
			END_IF
		END_IF
		actualPhi := ((fusionWeight-1) * actualPhi + AccPhi) /fusionWeight;
		(* error Zero crossing not handled !!! *)
	END_IF
	(* AccTheta is always accurate *)
	actualTheta := ((fusionWeight-1) * actualTheta + AccTheta) /fusionWeight;
END_IF

END_FUNCTION

// ---- POUs/Helping Functions/ATAN2_deg.TcPOU
FUNCTION ATAN2_deg : LREAL
VAR_INPUT	
    y : REAL; // y-coordinate
    x : REAL; // x-coordinate
END_VAR
VAR_OUTPUT
END_VAR

IF x > 0 THEN
    ATAN2_deg := ATAN(y / x);
ELSIF x < 0 AND y >= 0 THEN
    ATAN2_deg := ATAN(y / x) + pi;
ELSIF x < 0 AND y < 0 THEN
    ATAN2_deg := ATAN(y / x) - pi;
ELSIF x = 0 AND y > 0 THEN
    ATAN2_deg := pi / 2;
ELSIF x = 0 AND y < 0 THEN
    ATAN2_deg := -pi / 2;
ELSIF x = 0 AND y = 0 THEN
    ATAN2_deg := 0.0; // Undefined, but conventionally set to 0
END_IF

END_FUNCTION

// ---- POUs/Helping Functions/obsolete/iGetNextBufferPointer.TcPOU
FUNCTION iGetNextBufferPointer : INT
VAR_INPUT
	iBufferSize : INT;
	iActualPointerValue : INT;
END_VAR
VAR
	retVal : INT;
END_VAR

retVal := iActualPointerValue + 1;
IF retVal >= iBufferSize THEN retVal := 0; END_IF;
iGetNextBufferPointer := retVal;

END_FUNCTION

// ---- POUs/Helping Functions/obsolete/iGetPriorBufferPointer.TcPOU
FUNCTION iGetPriorBufferPointer : INT
VAR_INPUT
	iBufferSize : INT;
	iActualPointerValue : INT;
END_VAR
VAR
	retVal : INT;
END_VAR

retVal := iActualPointerValue - 1;
IF retVal < 0 THEN retVal := iBufferSize - 1; END_IF;
iGetPriorBufferPointer := retVal;

END_FUNCTION

// ---- GlobalTextList.TcGTLO
TEXTLIST GlobalTextList
  896 = '%.2f'
  216 = '%.3f'
  253 = '%d'
  460 = '%f'
  671 = 'Abgleich'
  162 = 'Accel X-Axis: %.0f'
  797 = 'Accel X-Axis: %.3f'
  669 = 'Accel Y-Axis: %.0f'
  525 = 'Accel Y-Axis: %.3f'
  265 = 'Accel Z-Axis: %.0f'
  89 = 'Accel Z-Axis: %.3f'
  553 = 'AccelY-Axis: %.0f'
  599 = 'Axis 1: %.3f'
  306 = 'Axis 2: %.3f'
  443 = 'Axis 3: %.3f'
  696 = 'Bytes: %d'
  819 = 'Calibrate'
  603 = 'Complementary'
  288 = 'Euler Angle Gamma%.3f'
  833 = 'Euler Angle Gamma: %.3f'
  868 = 'Euler Angle Phi: %.3f'
  3 = 'Euler Angle Psi%.3f'
  605 = 'Euler Angle Psi: %.3f'
  48 = 'Euler Angle Theta: %.3f'
  709 = 'Euler Angle: %.3f'
  626 = 'Euler Anlge Phi: %.3f'
  690 = 'Euler Anlge Theta: %.3f'
  952 = 'FThrh: %f'
  88 = 'FWeight: %f'
  277 = 'FWindow: %d'
  397 = 'Gyro X-Axis: %.0f'
  434 = 'Gyro X-Axis: %.3f'
  598 = 'Gyro Y-Axis: %.0f'
  123 = 'Gyro Y-Axis: %.3f'
  740 = 'Gyro Z-Axis: %.0f'
  955 = 'Gyro Z-Axis: %.3f'
  368 = 'Kalman'
  298 = 'Madgwick'
  943 = 'Mahony'
  68 = 'Phi: %.3f'
  223 = 'Psi: %.3f'
  666 = 'Read FIFO'
  614 = 'Reset'
  977 = 'Reset Angles'
  201 = 'Reset angles'
  848 = 'Reset Euler angles'
  850 = 'Reset Euler Angles'
  479 = 'Reset Winkel'
  983 = 'Set Angles to Zero'
  172 = 'Set Zero'
  221 = 'Set Zero Position'
  409 = 'Tara'
  233 = 'Theta: %.3f'
  2 = 'Use Sensorfusion'
  745 = 'Without Fusion'
  176 = 'X-Axis: %.0f'
  300 = 'X-Axis: %.0f mg'
  5 = 'X-Axis: %.0fmg'
  295 = 'X-Axis: %.3f'
  74 = 'X-Axis: %f mg'
  884 = 'X-Axis: %f.0 mg'
  794 = 'Y-Axis: %.0f'
  590 = 'Y-Axis: %.0fmg'
  132 = 'Y-Axis: %.3f'
  190 = 'Y-Axis: %f mg'
  637 = 'Y-Axis: %f.0 mg'
  272 = 'Z-Axis: %.0f'
  602 = 'Z-Axis: %.0fmg'
  518 = 'Z-Axis: %.3f'
  678 = 'Z-Axis: %f mg'
  248 = 'Z-Axis: %f.0 mg'
  142 = '°'
END_TEXTLIST

// ---- VISUs/Visualization.TcVIS
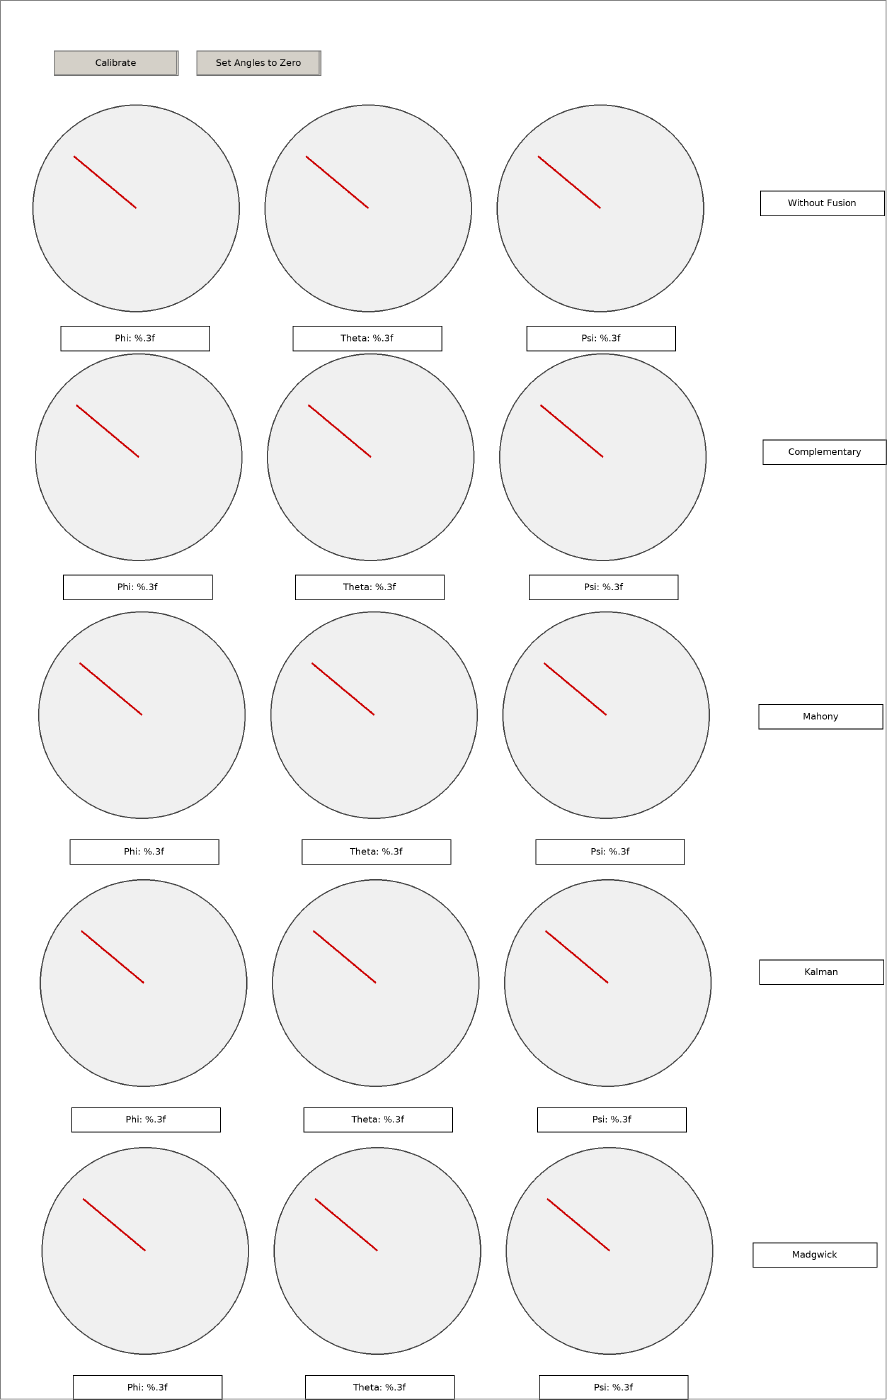
VISUALIZATION Visualization  // 1070x1688
    Button (65,61 150x30), "Calibrate", colour toggle: MAIN.bReady
        p2175578022: 16#FF808080
        p573394764: 16#FF80FF80
        tap MAIN.bReset
    Meter360 (42,426 250x250), value: MAIN.fbComplementaryFilter.stEulerAngle_deg.X, style: Meter-Meter360-Gray, scale format: %d, scale -180..180
        p518627256: °
    Meter360 (322,426 250x250), value: MAIN.fbComplementaryFilter.stEulerAngle_deg.Y, style: Meter-Meter360-Gray, scale format: %d, scale -180..180
        p518627256: °
    Meter360 (602,426 250x250), value: MAIN.fbComplementaryFilter.stEulerAngle_deg.Z, style: Meter-Meter360-Gray, scale format: %d, scale -180..180
        p518627256: °
    Rectangle (76,693 180x30), "Phi: %.3f", text variable: MAIN.fbComplementaryFilter.stEulerAngle_deg.X
    Rectangle (356,693 180x30), "Theta: %.3f", text variable: MAIN.fbComplementaryFilter.stEulerAngle_deg.Y
    Rectangle (638,693 180x30), "Psi: %.3f", text variable: MAIN.fbComplementaryFilter.stEulerAngle_deg.Z
    Meter360 (46,737 250x250), value: MAIN.fbMahonyFilter.stEulerAngle_deg.X, style: Meter-Meter360-Gray, scale format: %d, scale -180..180
        p518627256: °
    Meter360 (326,737 250x250), value: MAIN.fbMahonyFilter.stEulerAngle_deg.Y, style: Meter-Meter360-Gray, scale format: %d, scale -180..180
        p518627256: °
    Meter360 (606,737 250x250), value: MAIN.fbMahonyFilter.stEulerAngle_deg.Z, style: Meter-Meter360-Gray, scale format: %d, scale -180..180
        p518627256: °
    Rectangle (84,1012 180x30), "Phi: %.3f", text variable: MAIN.fbMahonyFilter.stEulerAngle_deg.X
    Rectangle (364,1012 180x30), "Theta: %.3f", text variable: MAIN.fbMahonyFilter.stEulerAngle_deg.Y
    Rectangle (646,1012 180x30), "Psi: %.3f", text variable: MAIN.fbMahonyFilter.stEulerAngle_deg.Z
    Meter360 (48,1060 250x250), value: MAIN.fbKalmanFilter.stEulerAngle_deg.X, style: Meter-Meter360-Gray, scale format: %d, scale -180..180
        p518627256: °
    Meter360 (328,1060 250x250), value: MAIN.fbKalmanFilter.stEulerAngle_deg.Y, style: Meter-Meter360-Gray, scale format: %d, scale -180..180
        p518627256: °
    Meter360 (608,1060 250x250), value: MAIN.fbKalmanFilter.stEulerAngle_deg.Z, style: Meter-Meter360-Gray, scale format: %d, scale -180..180
        p518627256: °
    Rectangle (86,1335 180x30), "Phi: %.3f", text variable: MAIN.fbKalmanFilter.stEulerAngle_deg.X
    Rectangle (366,1335 180x30), "Theta: %.3f", text variable: MAIN.fbKalmanFilter.stEulerAngle_deg.Y
    Rectangle (648,1335 180x30), "Psi: %.3f", text variable: MAIN.fbKalmanFilter.stEulerAngle_deg.Z
    Meter360 (50,1383 250x250), value: MAIN.fbMadgwickFilter.stEulerAngle_deg.X, style: Meter-Meter360-Gray, scale format: %d, scale -180..180
        p518627256: °
    Meter360 (330,1383 250x250), value: MAIN.fbMadgwickFilter.stEulerAngle_deg.Y, style: Meter-Meter360-Gray, scale format: %d, scale -180..180
        p518627256: °
    Meter360 (610,1383 250x250), value: MAIN.fbMadgwickFilter.stEulerAngle_deg.Z, style: Meter-Meter360-Gray, scale format: %d, scale -180..180
        p518627256: °
    Rectangle (88,1658 180x30), "Phi: %.3f", text variable: MAIN.fbMadgwickFilter.stEulerAngle_deg.X
    Rectangle (368,1658 180x30), "Theta: %.3f", text variable: MAIN.fbMadgwickFilter.stEulerAngle_deg.Y
    Rectangle (650,1658 180x30), "Psi: %.3f", text variable: MAIN.fbMadgwickFilter.stEulerAngle_deg.Z
    RoundedRectangle (920,530 150x30), "Complementary"
    RoundedRectangle (915,849 150x30), "Mahony"
    RoundedRectangle (916,1157 150x30), "Kalman"
    RoundedRectangle (908,1498 150x30), "Madgwick"
    Meter360 (39,126 250x250), value: MAIN.stEulerAngle_Gyro.X, style: Meter-Meter360-Gray, scale format: %d, scale -180..180
        p518627256: °
    Meter360 (319,126 250x250), value: MAIN.stEulerAngle_Gyro.Y, style: Meter-Meter360-Gray, scale format: %d, scale -180..180
        p518627256: °
    Meter360 (599,126 250x250), value: MAIN.stEulerAngle_Gyro.Z, style: Meter-Meter360-Gray, scale format: %d, scale -180..180
        p518627256: °
    Rectangle (73,393 180x30), "Phi: %.3f", text variable: MAIN.stEulerAngle_Gyro.X
    Rectangle (353,393 180x30), "Theta: %.3f", text variable: MAIN.stEulerAngle_Gyro.Y
    Rectangle (635,393 180x30), "Psi: %.3f", text variable: MAIN.stEulerAngle_Gyro.Z
    RoundedRectangle (917,230 150x30), "Without Fusion"
    Button (237,61 150x30), "Set Angles to Zero"
        tap MAIN.bResetAngles
END_VISUALIZATION
